# EPICS substitutions: db/EL1004.substitutions
file EL1004.template
{ 	pattern
	{
		TERMINAL,
		DESC1,	ZNAM1,	ONAM1,	ZSV1,	OSV1,	COSV1,	SCAN1,
		DESC2,	ZNAM2,	ONAM2,	ZSV2,	OSV2,	COSV2,	SCAN2,
		DESC3,	ZNAM3,	ONAM3,	ZSV3,	OSV3,	COSV3,	SCAN3,
		DESC4,	ZNAM4,	ONAM4,	ZSV4,	OSV4,	COSV4,	SCAN4
	}
	{
	}
}
